// TIA Portal V16 export
// export: Created 2023-03-29T11:04:27.3725246Z, ExportSetting WithDefaults, DisplayName Totally Integrated Automation Portal, DisplayVersion V16 Update 6, DisplayName TIA Portal Version Control Interface, DisplayVersion V16 Update 2, DisplayName TIA Portal Openness, DisplayVersion V16 Update 6, DisplayName STEP 7 Professional, DisplayVersion V16 Update 6, DisplayName STEP 7 Safety, DisplayVersion V16, DisplayName WinCC Advanced, DisplayVersion V16 Update 6
ORGANIZATION_BLOCK "Cyclic interrupt"   // OB30, LAD, CyclicInterrupt
{ S7_Optimized_Access := 'TRUE' }
AUTHOR : RTecmer
VERSION : 0.1
// stored: AutoNumber true, IsIECCheckEnabled false, SetENOAutomatically false
   VAR_TEMP
      Temp_SV_Int : Int;
      PV_Temp : Real;
      Temp_1 : Real;
   END_VAR
   VAR_TEMP   // added for the SCL form of the ladder/FBD networks
      _w1 : Bool;
      _w2 : Bool;
   END_VAR
BEGIN

REGION Network 1: WatchDog HMI
   // Do zrobienia
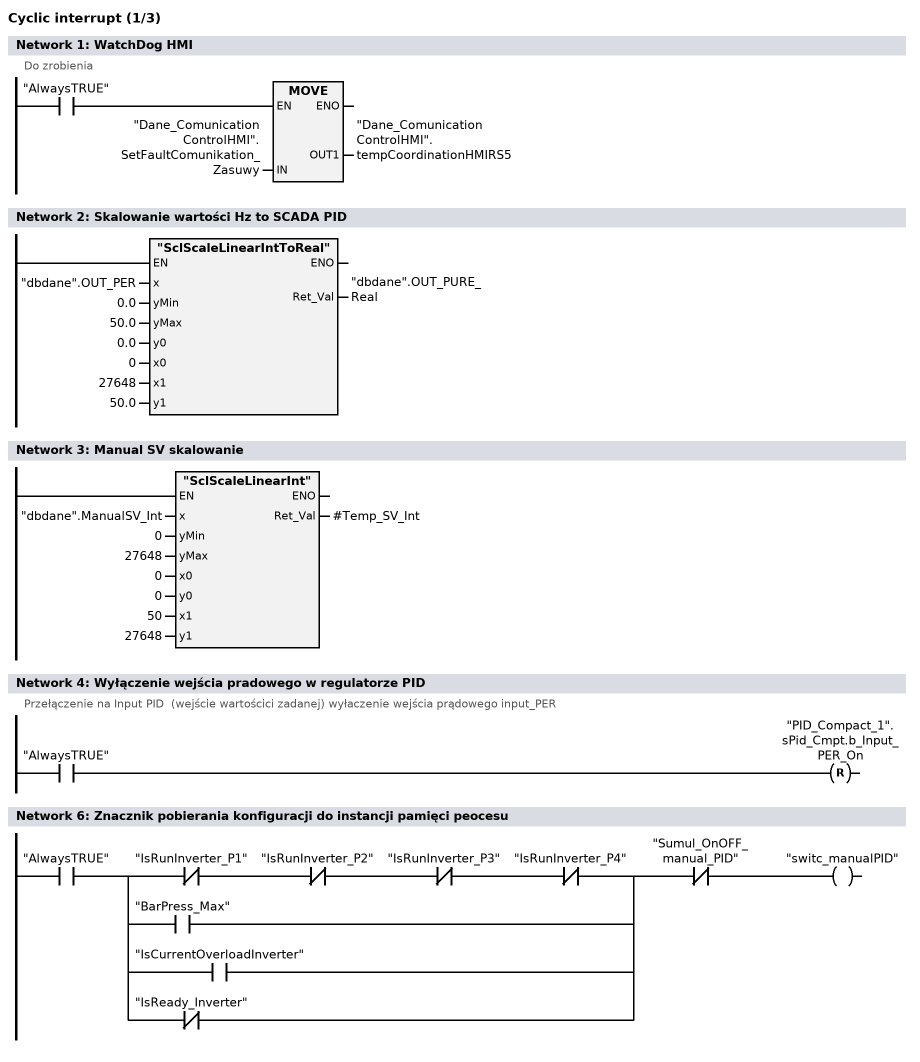
   RUNG wire#powerrail
      Contact( "AlwaysTRUE" )
      Move(in := "Dane_ComunicationControlHMI".SetFaultComunikation_Zasuwy, out1 => "Dane_ComunicationControlHMI".tempCoordinationHMIRS5)
   END_RUNG
   // the same network as SCL:
   IF "AlwaysTRUE" THEN
       "Dane_ComunicationControlHMI".tempCoordinationHMIRS5 := "Dane_ComunicationControlHMI".SetFaultComunikation_Zasuwy;
   END_IF;
END_REGION

REGION Network 2: Skalowanie wartości Hz to SCADA PID
   RUNG wire#powerrail
      "SclScaleLinearIntToReal"(x := "dbdane".OUT_PER, yMin := 0.0, yMax := 50.0, y0 := 0.0, x0 := 0, x1 := 27648, y1 := 50.0, Ret_Val => "dbdane".OUT_PURE_Real)
   END_RUNG
   // the same network as SCL:
   "dbdane".OUT_PURE_Real := "SclScaleLinearIntToReal"(x := "dbdane".OUT_PER,
                           yMin := 0.0,
                           yMax := 50.0,
                           y0 := 0.0,
                           x0 := 0,
                           x1 := 27648,
                           y1 := 50.0);
END_REGION

REGION Network 3: Manual SV skalowanie
   RUNG wire#powerrail
      "SclScaleLinearInt"(x := "dbdane".ManualSV_Int, yMin := 0, yMax := 27648, x0 := 0, y0 := 0, x1 := 50, y1 := 27648, Ret_Val => #Temp_SV_Int)
   END_RUNG
   // the same network as SCL:
   #Temp_SV_Int := "SclScaleLinearInt"(x := "dbdane".ManualSV_Int,
                           yMin := 0,
                           yMax := 27648,
                           x0 := 0,
                           y0 := 0,
                           x1 := 50,
                           y1 := 27648);
END_REGION

REGION Network 4: Wyłączenie wejścia pradowego w regulatorze PID
   // Przełączenie na Input PID  (wejście wartościci zadanej) wyłaczenie wejścia prądowego input_PER
   RUNG wire#powerrail
      Contact( "AlwaysTRUE" )
      R_Coil( "PID_Compact_1".sPid_Cmpt.b_Input_PER_On )
   END_RUNG
   // the same network as SCL:
   IF "AlwaysTRUE" THEN "PID_Compact_1".sPid_Cmpt.b_Input_PER_On := FALSE; END_IF;
END_REGION

REGION Network 5: Skalowanie wartośc pressure oxygen
   // Przetwornik ciśnienia (0-1bar) 
   // !!!!!! Znienić po zamontowaniu właściwego !!!!!!! 
   // obecnie czujnik 10 bar
END_REGION

REGION Network 6: Znacznik pobierania konfiguracji do instancji pamięci peocesu
   RUNG wire#powerrail
      Contact( "AlwaysTRUE" )
      wire#w1
      I_Contact( "IsRunInverter_P1" )
      I_Contact( "IsRunInverter_P2" )
      I_Contact( "IsRunInverter_P3" )
      I_Contact( "IsRunInverter_P4" )
      wire#w2
      I_Contact( "Sumul_OnOFF_manual_PID" )
      Coil( "switc_manualPID" )
   END_RUNG
   RUNG wire#w1
      Contact( "BarPress_Max" )
   END_RUNG wire#w2
   RUNG wire#w1
      Contact( "IsCurrentOverloadInverter" )
   END_RUNG wire#w2
   RUNG wire#w1
      I_Contact( "IsReady_Inverter" )
   END_RUNG wire#w2
   // the same network as SCL:
   "switc_manualPID" := "AlwaysTRUE" AND ((NOT "IsRunInverter_P1" AND NOT "IsRunInverter_P2" AND NOT "IsRunInverter_P3" AND NOT "IsRunInverter_P4") OR "BarPress_Max" OR "IsCurrentOverloadInverter" OR NOT "IsReady_Inverter") AND NOT "Sumul_OnOFF_manual_PID";
END_REGION

REGION Network 7: PID
   // Linia załączenia Manual wykonyje zadanie przekazania wartości minimalnej gdy nie pracuje falownik.
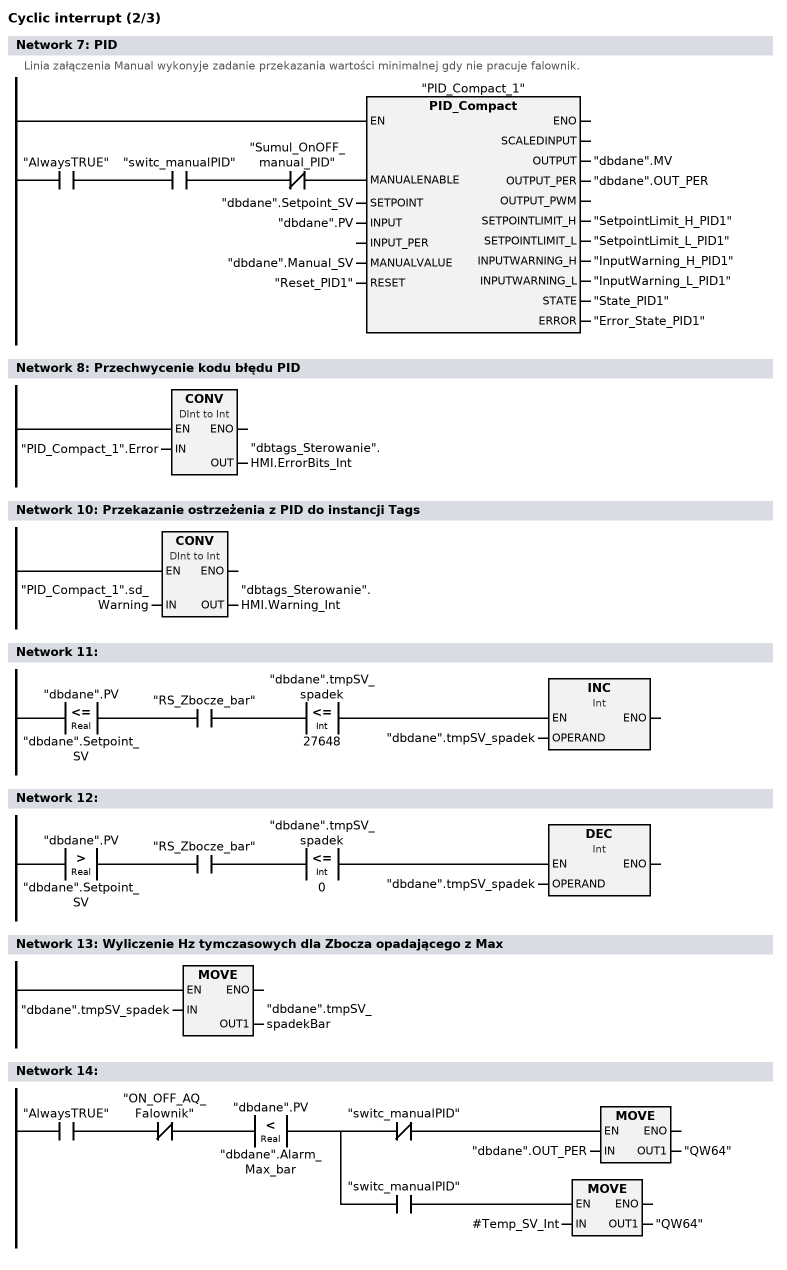
   RUNG wire#powerrail
      "PID_Compact_1".PID_Compact(ManualEnable := wire#w1, Setpoint := "dbdane".Setpoint_SV, Input := "dbdane".PV, Input_PER :=, ManualValue := "dbdane".Manual_SV, Reset := "Reset_PID1", ScaledInput =>, Output => "dbdane".MV, Output_PER => "dbdane".OUT_PER, Output_PWM =>, SetpointLimit_H => "SetpointLimit_H_PID1", SetpointLimit_L => "SetpointLimit_L_PID1", InputWarning_H => "InputWarning_H_PID1", InputWarning_L => "InputWarning_L_PID1", State => "State_PID1", Error => "Error_State_PID1")
   END_RUNG
   RUNG wire#powerrail
      Contact( "AlwaysTRUE" )
      Contact( "switc_manualPID" )
      I_Contact( "Sumul_OnOFF_manual_PID" )
   END_RUNG wire#w1
   // the same network as SCL:
   "PID_Compact_1"(ManualEnable := "AlwaysTRUE" AND "switc_manualPID" AND NOT "Sumul_OnOFF_manual_PID",   // PID_Compact
                   Setpoint := "dbdane".Setpoint_SV,
                   Input := "dbdane".PV,
                   ManualValue := "dbdane".Manual_SV,
                   Reset := "Reset_PID1",
                   Output => "dbdane".MV,
                   Output_PER => "dbdane".OUT_PER,
                   SetpointLimit_H => "SetpointLimit_H_PID1",
                   SetpointLimit_L => "SetpointLimit_L_PID1",
                   InputWarning_H => "InputWarning_H_PID1",
                   InputWarning_L => "InputWarning_L_PID1",
                   State => "State_PID1",
                   Error => "Error_State_PID1");
END_REGION

REGION Network 8: Przechwycenie kodu błędu PID
   RUNG wire#powerrail
      { S7_Templates := "[SrcType := DInt, DestType := Int]"; S7_GenerateENO := "TRUE" } Convert(in := "PID_Compact_1".Error, out => "dbtags_Sterowanie".HMI.ErrorBits_Int)
   END_RUNG
   // the same network as SCL:
   "dbtags_Sterowanie".HMI.ErrorBits_Int := DINT_TO_INT("PID_Compact_1".Error);
END_REGION

REGION Network 10: Przekazanie ostrzeżenia z PID do instancji Tags
   RUNG wire#powerrail
      { S7_Templates := "[SrcType := DInt, DestType := Int]"; S7_GenerateENO := "TRUE" } Convert(in := "PID_Compact_1".sd_Warning, out => "dbtags_Sterowanie".HMI.Warning_Int)
   END_RUNG
   // the same network as SCL:
   "dbtags_Sterowanie".HMI.Warning_Int := DINT_TO_INT("PID_Compact_1".sd_Warning);
END_REGION

REGION Network 11
   RUNG wire#powerrail
      { S7_Templates := "SrcType := Real" } LE_Contact(in1 := "dbdane".PV, in2 := "dbdane".Setpoint_SV)
      Contact( "RS_Zbocze_bar" )
      { S7_Templates := "SrcType := Int" } LE_Contact(in1 := "dbdane".tmpSV_spadek, in2 := 27648)
      { S7_Templates := "DestType := Int" } Inc( "dbdane".tmpSV_spadek )
   END_RUNG
   // the same network as SCL:
   IF ("dbdane".PV <= "dbdane".Setpoint_SV) AND "RS_Zbocze_bar" AND ("dbdane".tmpSV_spadek <= 27648) THEN
       "dbdane".tmpSV_spadek := "dbdane".tmpSV_spadek + 1;
   END_IF;
END_REGION

REGION Network 12
   RUNG wire#powerrail
      { S7_Templates := "SrcType := Real" } GT_Contact(in1 := "dbdane".PV, in2 := "dbdane".Setpoint_SV)
      Contact( "RS_Zbocze_bar" )
      { S7_Templates := "SrcType := Int" } LE_Contact(in1 := "dbdane".tmpSV_spadek, in2 := 0)
      { S7_Templates := "DestType := Int" } Dec( "dbdane".tmpSV_spadek )
   END_RUNG
   // the same network as SCL:
   IF ("dbdane".PV > "dbdane".Setpoint_SV) AND "RS_Zbocze_bar" AND ("dbdane".tmpSV_spadek <= 0) THEN
       "dbdane".tmpSV_spadek := "dbdane".tmpSV_spadek - 1;
   END_IF;
END_REGION

REGION Network 13: Wyliczenie Hz tymczasowych dla Zbocza opadającego z Max
   RUNG wire#powerrail
      Move(in := "dbdane".tmpSV_spadek, out1 => "dbdane".tmpSV_spadekBar)
   END_RUNG
   // the same network as SCL:
   "dbdane".tmpSV_spadekBar := "dbdane".tmpSV_spadek;
END_REGION

REGION Network 14
   RUNG wire#powerrail
      Contact( "AlwaysTRUE" )
      I_Contact( "ON_OFF_AQ_Falownik" )
      { S7_Templates := "SrcType := Real" } LT_Contact(in1 := "dbdane".PV, in2 := "dbdane".Alarm_Max_bar)
      wire#w1
      I_Contact( "switc_manualPID" )
      { S7_GenerateENO := "TRUE" } Move(in := "dbdane".OUT_PER, out1 => "QW64")
   END_RUNG
   RUNG wire#w1
      Contact( "switc_manualPID" )
      { S7_GenerateENO := "TRUE" } Move(in := #Temp_SV_Int, out1 => "QW64")
   END_RUNG
   // the same network as SCL:
   #_w1 := "AlwaysTRUE" AND NOT "ON_OFF_AQ_Falownik" AND ("dbdane".PV < "dbdane".Alarm_Max_bar);
   IF #_w1 AND NOT "switc_manualPID" THEN "QW64" := "dbdane".OUT_PER; END_IF;
   IF #_w1 AND "switc_manualPID" THEN "QW64" := #Temp_SV_Int; END_IF;
END_REGION

REGION Network 15: Wyłączenie regulacji Hz
   // Jeśli ciśnienie alarmowe ustawienie na wyjściu Hz = 0
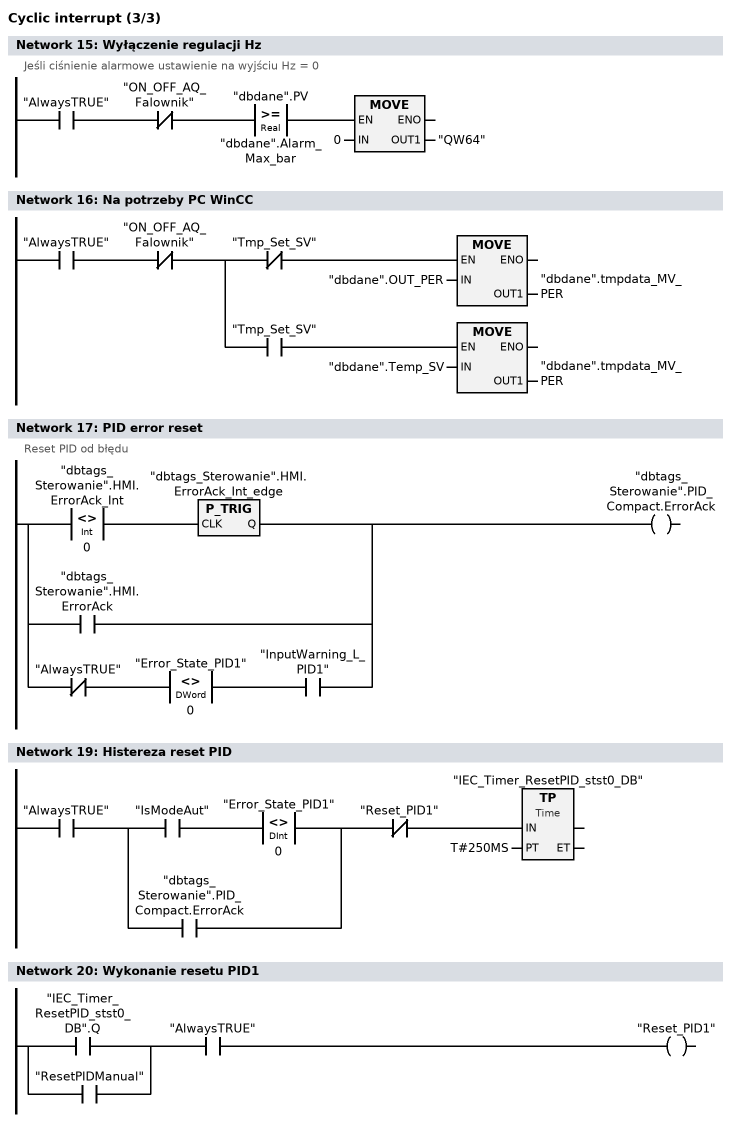
   RUNG wire#powerrail
      Contact( "AlwaysTRUE" )
      I_Contact( "ON_OFF_AQ_Falownik" )
      { S7_Templates := "SrcType := Real" } GE_Contact(in1 := "dbdane".PV, in2 := "dbdane".Alarm_Max_bar)
      { S7_GenerateENO := "TRUE" } Move(in := 0, out1 => "QW64")
   END_RUNG
   // the same network as SCL:
   IF "AlwaysTRUE" AND NOT "ON_OFF_AQ_Falownik" AND ("dbdane".PV >= "dbdane".Alarm_Max_bar) THEN
       "QW64" := 0;
   END_IF;
END_REGION

REGION Network 16: Na potrzeby PC WinCC
   RUNG wire#powerrail
      Contact( "AlwaysTRUE" )
      I_Contact( "ON_OFF_AQ_Falownik" )
      wire#w1
      I_Contact( "Tmp_Set_SV" )
      { S7_GenerateENO := "TRUE" } Move(in := "dbdane".OUT_PER, out1 => "dbdane".tmpdata_MV_PER)
   END_RUNG
   RUNG wire#w1
      Contact( "Tmp_Set_SV" )
      { S7_GenerateENO := "TRUE" } Move(in := "dbdane".Temp_SV, out1 => "dbdane".tmpdata_MV_PER)
   END_RUNG
   // the same network as SCL:
   #_w1 := "AlwaysTRUE" AND NOT "ON_OFF_AQ_Falownik";
   IF #_w1 AND NOT "Tmp_Set_SV" THEN "dbdane".tmpdata_MV_PER := "dbdane".OUT_PER; END_IF;
   IF #_w1 AND "Tmp_Set_SV" THEN "dbdane".tmpdata_MV_PER := "dbdane".Temp_SV; END_IF;
END_REGION

REGION Network 17: PID error reset
   // Reset PID od błędu
   RUNG wire#powerrail
      { S7_Templates := "SrcType := Int" } NE_Contact(in1 := "dbtags_Sterowanie".HMI.ErrorAck_Int, in2 := 0)
      P_Trig( "dbtags_Sterowanie".HMI.ErrorAck_Int_edge )
      wire#w1
      Coil( "dbtags_Sterowanie".PID_Compact.ErrorAck )
   END_RUNG
   RUNG wire#powerrail
      Contact( "dbtags_Sterowanie".HMI.ErrorAck )
   END_RUNG wire#w1
   RUNG wire#powerrail
      I_Contact( "AlwaysTRUE" )
      { S7_Templates := "SrcType := DWord" } NE_Contact(in1 := "Error_State_PID1", in2 := 0)
      Contact( "InputWarning_L_PID1" )
   END_RUNG wire#w1
   // the same network as SCL:
   #_w1 := "dbtags_Sterowanie".HMI.ErrorAck_Int <> 0;
   #_w2 := #_w1 AND NOT "dbtags_Sterowanie".HMI.ErrorAck_Int_edge;   // rising edge
   "dbtags_Sterowanie".HMI.ErrorAck_Int_edge := #_w1;
   "dbtags_Sterowanie".PID_Compact.ErrorAck := #_w2 OR "dbtags_Sterowanie".HMI.ErrorAck OR (NOT "AlwaysTRUE" AND ("Error_State_PID1" <> 0) AND "InputWarning_L_PID1");
END_REGION

REGION Network 19: Histereza reset PID
   RUNG wire#powerrail
      Contact( "AlwaysTRUE" )
      wire#w1
      Contact( "IsModeAut" )
      { S7_Templates := "SrcType := DInt" } NE_Contact(in1 := "Error_State_PID1", in2 := 0)
      wire#w2
      I_Contact( "Reset_PID1" )
      { S7_Templates := "time_type := Time" } "IEC_Timer_ResetPID_stst0_DB".TP(pt := T#250MS, et =>)
   END_RUNG
   RUNG wire#w1
      Contact( "dbtags_Sterowanie".PID_Compact.ErrorAck )
   END_RUNG wire#w2
   // the same network as SCL:
   "IEC_Timer_ResetPID_stst0_DB".TP(IN := "AlwaysTRUE" AND (("IsModeAut" AND ("Error_State_PID1" <> 0)) OR "dbtags_Sterowanie".PID_Compact.ErrorAck) AND NOT "Reset_PID1",
                           PT := T#250MS);
END_REGION

REGION Network 20: Wykonanie resetu PID1
   RUNG wire#powerrail
      Contact( "IEC_Timer_ResetPID_stst0_DB".Q )
      wire#w1
      Contact( "AlwaysTRUE" )
      Coil( "Reset_PID1" )
   END_RUNG
   RUNG wire#powerrail
      Contact( "ResetPIDManual" )
   END_RUNG wire#w1
   // the same network as SCL:
   "Reset_PID1" := ("IEC_Timer_ResetPID_stst0_DB".Q OR "ResetPIDManual") AND "AlwaysTRUE";
END_REGION
END_ORGANIZATION_BLOCK
